FUNCTION_BLOCK FB_ButtonEnable
VAR_INPUT
	SET:	BOOL;
	RESET:	BOOL;
END_VAR
VAR_IN_OUT
	Q: BOOL;
END_VAR
VAR
	trigger:	R_TRIG;
//	ftrigger:	F_TRIG;
END_VAR

trigger(CLK := SET);
//ftrigger(CLK := SET);

// if button was triggered, flip the state of the output
IF trigger.Q THEN
	Q := NOT Q;
END_IF

// if reset is enabled we disable the output
IF RESET THEN
	Q := FALSE;
END_IF

END_FUNCTION_BLOCK

(* stored: Version 1.1.0.1, ProductVersion 3.1.4024.15
   POU FB_ButtonEnable: Id {3211ceeb-9597-41c3-8547-3ce80543891d}, SpecialFunc None *)
